{attribute 'qualified_only'}
{attribute 'strict'}
{attribute 'to_string'}
TYPE eTcaTrolleyCmd :
(
	noCmd := 0,
	FillTrolley,
	RemoveTrolley,
	EmptyTrolley
);
END_TYPE

(* stored: Version 1.1.0.1
   DUT eTcaTrolleyCmd: Id {2c6c198f-4b5b-4094-83d5-14b539057647} *)
